FUNCTION RemoveIndexFromStringArray : BOOL
VAR_IN_OUT
	arr : ARRAY[*] OF STRING; //must start from 0 index
END_VAR
VAR_INPUT
	index : DINT;
END_VAR
VAR_OUTPUT
	numElements : DINT;
	nextIndex : DINT;
END_VAR
VAR
	i : DINT;
END_VAR

IF i < LOWER_BOUND(arr, 1) OR i > UPPER_BOUND(arr, 1) THEN
	RETURN;
END_IF

FOR i:=index TO UPPER_BOUND(arr, 1)-1 BY 1 DO
	arr[i] := arr[i+1];
END_FOR

arr[UPPER_BOUND(arr, 1)] := '';

RemoveIndexFromStringArray := TRUE;

END_FUNCTION

(* stored: Version 1.1.0.1, ProductVersion 3.1.4024.11
   POU RemoveIndexFromStringArray: Id {10c78833-0e22-41ff-bd79-d0cd734e6b2c}, SpecialFunc None *)
